{attribute 'GeneratedUsingTerminal: EL3351-0000-0016'}
{attribute addProperty BoxType "EL3351-0000-0016"}
{attribute addProperty Id "UnderrangeAT %I*BOOL1OverrangeAT %I*BOOL1ErrorAT %I*BOOL1TxPDO_StateAT %I*BOOL1TxPDO_ToggleAT %I*BOOL1ValueAT %I*DINT4"}
{attribute addProperty CRC "1432003048"}
{attribute addProperty Size "9"}
TYPE AISupply_Inputs_555AA1E8 :
STRUCT
	{attribute addProperty Name "Underrange"}
	Underrange AT %I* : BOOL;
	{attribute addProperty Name "Overrange"}
	Overrange AT %I* : BOOL;
	{attribute addProperty Name "Error"}
	Error AT %I* : BOOL;
	{attribute addProperty Name "TxPDO_State"}
	TxPDO_State AT %I* : BOOL;
	{attribute addProperty Name "TxPDO_Toggle"}
	TxPDO_Toggle AT %I* : BOOL;
	{attribute addProperty Name "Value"}
	Value AT %I* : DINT;
END_STRUCT
END_TYPE

(* stored: Version 1.2.0.0, ProductVersion 3.1.4024.9
   DUT AISupply_Inputs_555AA1E8: Id {e975d334-be54-4501-81ff-d97a073643db} *)
